FUNCTION_BLOCK RecordableStation001 EXTENDS TcoCore.TcoContext
VAR
    _components : RecordableStation001_Components(THIS^);
    _sequence : RecordableStation001_Sequencer(THIS^, eRestoreMode.None);
    _serviceModeTask : TcoCore.TcoTask(THIS^);
    _automatModeTask : TcoCore.TcoTask(THIS^);
END_VAR

(*~
    <docu>
        <summary>
            Main method of the TcoContext. This is the entry point of any control logic that belongs to this context.
            The call of this method is ensured by calling the <c>InstanceName.Run()</c> method, and it must not be called explicitly.
            This method is abstract, and it must be overridden in derived block.
        </summary>
    </docu>
~*)
METHOD PROTECTED Main
_sequence(components := _components);
_components();

IF (_serviceModeTask.Execute()) THEN
    _automatModeTask.Restore();
    _components.Service();
END_IF;

IF (_automatModeTask.Execute()) THEN
    _serviceModeTask.Restore();
    _sequence.Run();
END_IF;
END_METHOD

END_FUNCTION_BLOCK

(* stored: Version 1.1.0.1
   POU RecordableStation001: Id {d8716088-3f58-05d3-3548-fce641607337}, SpecialFunc None
   Method Main: Id {a859f906-ea2c-0da9-0be2-e7f4df0f11d5} *)
